// TIA Portal V16 export
// export: Created 2021-07-12T14:47:21.0947076Z, ExportSetting WithDefaults, DisplayName Totally Integrated Automation Portal, DisplayVersion V16, DisplayName TIA Portal Version Control Interface, DisplayVersion V16, DisplayName TIA Portal Openness, DisplayVersion V16, DisplayName STEP 7 Professional, DisplayVersion V16, DisplayName STEP 7 Safety, DisplayVersion V16, DisplayName WinCC Professional, DisplayVersion V16
TYPE "SimaHydTO_typeHMIConnectionVCharSelectorStatus"
TITLE = SimaHydTO_typeHMIConnectionVCharSelectorStatus
// HMI interface: Hydraulic characteristics (VChar) selection of VChar array - Status (PLC -> HMI)
// stored: IsFailsafeCompliant false
   STRUCT
      actualVCharIndex : Int;   // Actual selected array index
      selectedVCharInteger : UInt;   // DB number of actual selected valve characteristics as integer value
      selectedVChar : DB_ANY;   // DB number of actual selected valve characteristics
      selectedVCharName : WString[24];   // Name of actual selected valve characteristics
      dataValid : Bool;   // Selected data valid
      dataError : Bool;   // Error of data selection
   END_STRUCT;
END_TYPE
